// TIA Portal V20 export
DATA_BLOCK "SBK04"   // DB319
// stored: MemoryReserve 100
   VAR
      "GATE EC U/W MAIN PB.LOCK" : Bool := FALSE;
      "GATE EC U/W MAIN PB.RESET" : Bool := FALSE;
      SPARE : Bool := FALSE;
      SPARE_1 : Bool := FALSE;
      "GATE EC U/W MAIN PB.UNLOCK" : Bool := FALSE;
      SPARE_2 : Bool := FALSE;
      SPARE_3 : Bool := FALSE;
      SPARE_4 : Bool := FALSE;
      "GATE EC U/W MAIN PL.LOCK" : Bool := TRUE;
      "GATE EC U/W MAIN PL.UNLOCK" : Bool := FALSE;
      "GATE EC U/W MAIN PL.RESET" : Bool := TRUE;
   END_VAR
BEGIN
END_DATA_BLOCK
